FUNCTION_BLOCK UA_UnitIds (* OPC UA node IDs of the unit facade, below UaRoot *)
  (* Standard: 61499-2 *)
  (* Version 2.0, 2026-09-27, Project contributors, Filling cell reference model *)
  PACKAGE fillingcell;
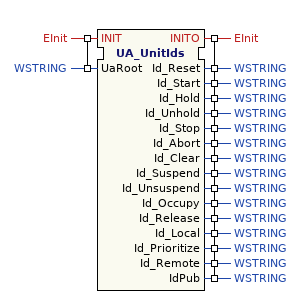
  EVENT_INPUT
    INIT : EInit WITH UaRoot;
  END_EVENT
  EVENT_OUTPUT
    INITO : EInit WITH Id_Reset, Id_Start, Id_Hold, Id_Unhold, Id_Stop, Id_Abort, Id_Clear, Id_Suspend, Id_Unsuspend, Id_Occupy, Id_Release, Id_Local, Id_Prioritize, Id_Remote, IdPub;
  END_EVENT
  VAR_INPUT
    UaRoot : WSTRING;
  END_VAR
  VAR_OUTPUT
    Id_Reset : WSTRING;
    Id_Start : WSTRING;
    Id_Hold : WSTRING;
    Id_Unhold : WSTRING;
    Id_Stop : WSTRING;
    Id_Abort : WSTRING;
    Id_Clear : WSTRING;
    Id_Suspend : WSTRING;
    Id_Unsuspend : WSTRING;
    Id_Occupy : WSTRING;
    Id_Release : WSTRING;
    Id_Local : WSTRING;
    Id_Prioritize : WSTRING;
    Id_Remote : WSTRING;
    IdPub : WSTRING;
  END_VAR
  EC_STATES
    INIT : INIT -> INITO;
  END_STATES
  ALGORITHM INIT IN ST:
Id_Reset := CONCAT(CONCAT("opc_ua[CREATE_METHOD;", UaRoot), "/Unit/Reset]");
Id_Start := CONCAT(CONCAT("opc_ua[CREATE_METHOD;", UaRoot), "/Unit/Start]");
Id_Hold := CONCAT(CONCAT("opc_ua[CREATE_METHOD;", UaRoot), "/Unit/Hold]");
Id_Unhold := CONCAT(CONCAT("opc_ua[CREATE_METHOD;", UaRoot), "/Unit/Unhold]");
Id_Stop := CONCAT(CONCAT("opc_ua[CREATE_METHOD;", UaRoot), "/Unit/Stop]");
Id_Abort := CONCAT(CONCAT("opc_ua[CREATE_METHOD;", UaRoot), "/Unit/Abort]");
Id_Clear := CONCAT(CONCAT("opc_ua[CREATE_METHOD;", UaRoot), "/Unit/Clear]");
Id_Suspend := CONCAT(CONCAT("opc_ua[CREATE_METHOD;", UaRoot), "/Unit/Suspend]");
Id_Unsuspend := CONCAT(CONCAT("opc_ua[CREATE_METHOD;", UaRoot), "/Unit/Unsuspend]");
Id_Occupy := CONCAT(CONCAT("opc_ua[CREATE_METHOD;", UaRoot), "/Occupation/Occupy]");
Id_Release := CONCAT(CONCAT("opc_ua[CREATE_METHOD;", UaRoot), "/Occupation/Release]");
Id_Local := CONCAT(CONCAT("opc_ua[CREATE_METHOD;", UaRoot), "/Occupation/Local]");
Id_Prioritize := CONCAT(CONCAT("opc_ua[CREATE_METHOD;", UaRoot), "/Occupation/Prioritize]");
Id_Remote := CONCAT(CONCAT("opc_ua[CREATE_METHOD;", UaRoot), "/Occupation/Remote]");
IdPub := CONCAT(CONCAT(CONCAT(CONCAT(CONCAT(CONCAT(CONCAT(CONCAT("opc_ua[WRITE;", UaRoot), "/Unit/State;"), UaRoot), "/Unit/Mode;"), UaRoot), "/Occupation/State;"), UaRoot), "/Occupation/Owner]");
  END_ALGORITHM
END_FUNCTION_BLOCK
